FUNCTION_BLOCK FB_FMS205_Test
VAR_INPUT
	TestAlimentador: BOOL;
END_VAR
VAR_OUTPUT
END_VAR
VAR
END_VAR

END_FUNCTION_BLOCK

(* stored: Version 1.1.0.1, ProductVersion 3.1.4024.11
   POU FB_FMS205_Test: Id {eca8bbf9-f875-4e8d-a3b2-e4a2d2dcccf7}, SpecialFunc None *)
